// Mitsubishi GX Works2 project: 0709계산기교과서   PLC: Q02/Q02H

PROGRAM MAIN
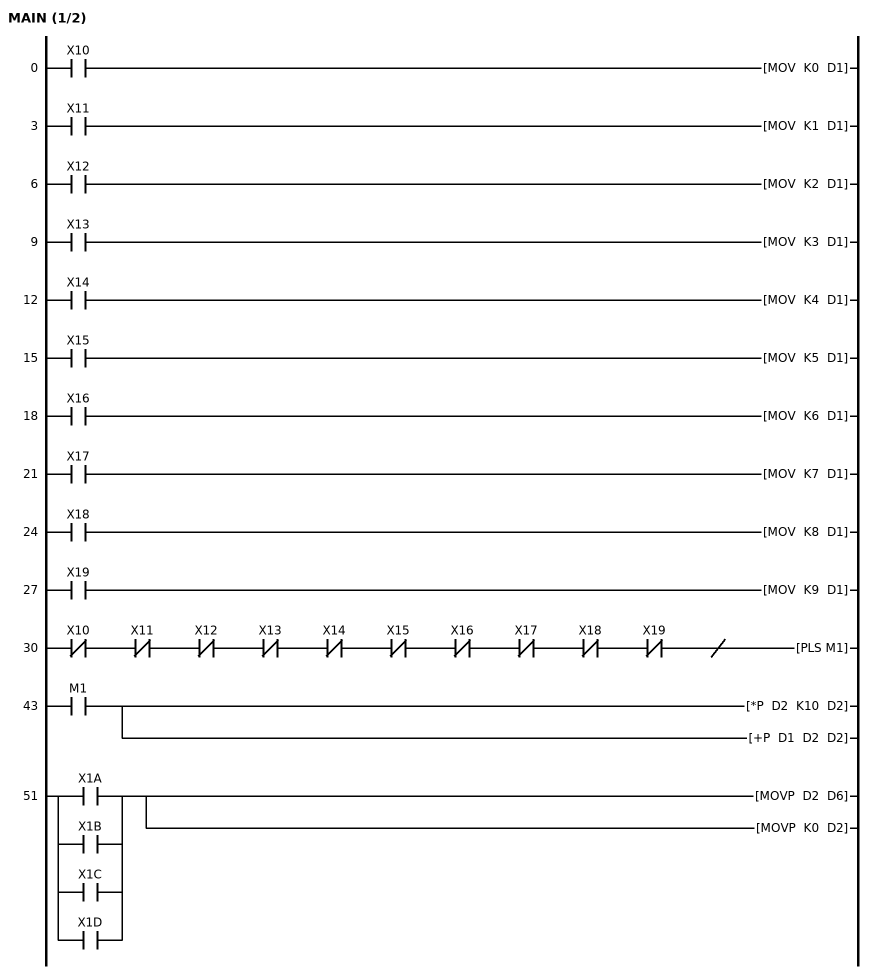
0     LD      X10
      MOV     K0 D1
3     LD      X11
      MOV     K1 D1
6     LD      X12
      MOV     K2 D1
9     LD      X13
      MOV     K3 D1
12    LD      X14
      MOV     K4 D1
15    LD      X15
      MOV     K5 D1
18    LD      X16
      MOV     K6 D1
21    LD      X17
      MOV     K7 D1
24    LD      X18
      MOV     K8 D1
27    LD      X19
      MOV     K9 D1
30    LDI     X10
      ANI     X11
      ANI     X12
      ANI     X13
      ANI     X14
      ANI     X15
      ANI     X16
      ANI     X17
      ANI     X18
      ANI     X19
      INV
      PLS     M1
43    LD      M1
      *P      D2 K10 D2
      +P      D1 D2 D2
51    LD      X1A
      OR      X1B
      OR      X1C
      OR      X1D
      MOVP    D2 D6
      MOVP    K0 D2
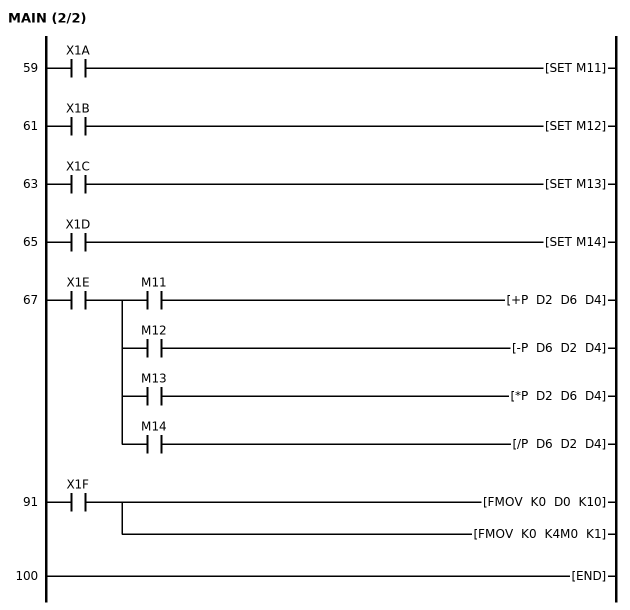
59    LD      X1A
      SET     M11
61    LD      X1B
      SET     M12
63    LD      X1C
      SET     M13
65    LD      X1D
      SET     M14
67    LD      X1E
      MPS
      AND     M11
      +P      D2 D6 D4
      MRD
      AND     M12
      -P      D6 D2 D4
      MRD
      AND     M13
      *P      D2 D6 D4
      MPP
      AND     M14
      /P      D6 D2 D4
91    LD      X1F
      FMOV    K0 D0 K10
      FMOV    K0 K4M0 K1
100   END
END_PROGRAM
